FUNCTION F_Square : REAL
VAR_INPUT
	ymin	: REAL;	// Minimalwert
	ymax	: REAL;	// Maximalwert
	yoff	: REAL; // offset
	w		: REAL; // Kreisfrequenz (rad/s)
	t		: REAL; // Time (s)
END_VAR
VAR
	sinRes	: REAL; // sine result
	squareRes: REAL;
END_VAR

sinRes := SIN(w*t);

IF (sinRes > 0) THEN
	squareRes := ymin;
ELSE
	squareRes := ymax;
END_IF

F_Square := squareRes + yoff;

END_FUNCTION

(* stored: Version 1.1.0.1, ProductVersion 3.1.4024.9
   POU F_Square: Id {ce683447-e8cf-4378-bff1-06638e6e9c36}, SpecialFunc None *)
